# EPICS autosave request: iocBoot/iocProsilica/auto_settings.req
file "ADBase_settings.req",  P=$(P),  D=cam1:
file "NDStdArrays_settings.req", P=$(P),  A=image1:
file "ADFile_settings.req",  P=$(P),  F=file1:
